PROGRAM MAIN
VAR
	state : (IDLE, FIND_FILES, GET_FILES, DONE) := IDLE;
	
	fileCollection : FileSystemEntryCollection;
	fileFinder : FileFinder(fileCollection);
	searchPath : T_MaxString := 'C:\dev\vision-toolkit\test\integration\';
	fileSystemEntry : I_FileSystemEntry;
	path : T_MaxString;
	
END_VAR

// find files in supplied initial folder & sub-folders and populate a collection.

CASE state OF 
	
	IDLE : //
	
	FIND_FILES:
	
		IF (fileFinder.Find(searchPath, '*.tcgraph')) THEN
			state := GET_FILES;
			
		END_IF
	
	GET_FILES:
	
		fileSystemEntry := fileCollection.GetFirst();
		WHILE (NOT fileSystemEntry.IsNull) DO

			path := fileSystemEntry.Path;
			fileSystemEntry := fileCollection.GetNext(fileSystemEntry);
			
		END_WHILE
		fileCollection.Clear();
		
		state := DONE;
		
	DONE: //
	
END_CASE

END_PROGRAM

(* stored: Version 1.1.0.1, ProductVersion 3.1.4024.9
   POU MAIN: Id {ec38523b-9156-4770-8e81-c6221898da8f}, SpecialFunc None *)
